FUNCTION F_PHYS_LREAL_TO_RAW (* Convert physical LREAL value to ISOBUS raw UDINT. ISOBUS formula: display = (raw + offset) * scale Inverse:        raw     = UDINT(DINT(phys / scale) - offset) Example: phys=-500.0, scale=0.01, offset=-100000 DINT(-500.0 / 0.01) = -50000 -50000 - (-100000)  = 50000 UDINT(50000)        = 50000  -> UT displays (50000 + (-100000)) 0.01 = -500.00 *)
  (* Standard: 61499-2; Description: Copyright (c) 2026 Meisterschulen am Ostbahnhof This program and the accompanying materials are made available under the terms of the Eclipse Public License 2.0 which is available at https://www.eclipse.org/legal/epl-2.0/ SPDX-License-Identifier: EPL-2.0 *)
  (* Version 1.0, 2026-04-21, Franz Höpfinger, Meisterschulen am Ostbahnhof *)
  PACKAGE logiBUS::utils::conversion::phys;
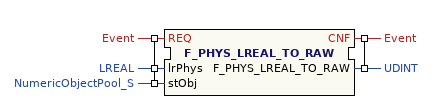
  EVENT_INPUT
    REQ WITH lrPhys, stObj;
  END_EVENT
  EVENT_OUTPUT
    CNF WITH F_PHYS_LREAL_TO_RAW;
  END_EVENT
  VAR_INPUT
    lrPhys : LREAL;
    stObj : logiBUS::utils::conversion::phys::NumericObjectPool_S;
  END_VAR
  VAR_OUTPUT
    F_PHYS_LREAL_TO_RAW : UDINT;
  END_VAR
  BODY IN ST:
PACKAGE logiBUS::utils::conversion::phys;

(* Convert physical LREAL value to ISOBUS raw UDINT.
 * ISOBUS formula: display = (raw + offset) * scale Inverse:        raw     = UDINT(DINT(phys /
 * scale) - offset)
 * *
 * Example: phys=-500.0, scale=0.01, offset=-100000 DINT(-500.0 / 0.01) = -50000
 * -50000 - (-100000)  = 50000 UDINT(50000)        = 50000  -> UT displays (50000 + (-100000)) *
 * 0.01 = -500.00 *)
FUNCTION F_PHYS_LREAL_TO_RAW : UDINT

VAR_INPUT
	lrPhys : LREAL;
	stObj : NumericObjectPool_S;
END_VAR

F_PHYS_LREAL_TO_RAW := DINT_TO_UDINT(LREAL_TO_DINT(lrPhys / stObj.r32Scale) - stObj.i32Offset);

END_FUNCTION
  END_BODY
END_FUNCTION
